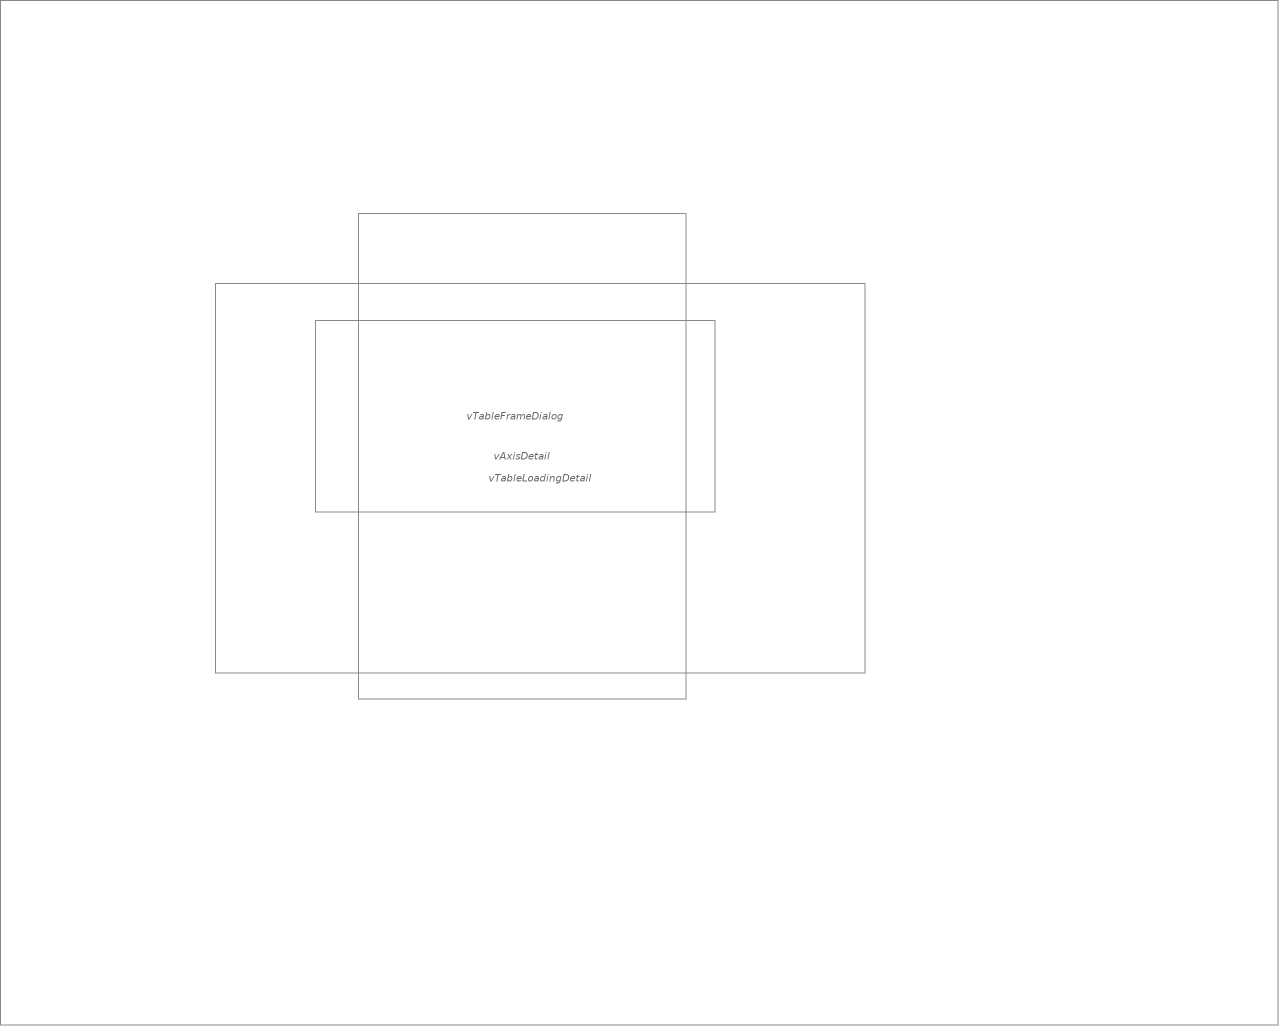
VISUALIZATION vWeighingTunnel  // 1279x1026
VAR_IN_OUT
	fbTableControl: FB_TableControl;
END_VAR
    Rectangle (19,221 146x45), "Drawer Unlock Request", colour toggle: MAIN.fbWeighingStation.bDrawerUnlockRequest, input disabled if: MAIN.fbWeighingStation.stSettings.iMaxNOK_Bottles = MAIN.fbWeighingStation.stSettings.iNOK_BottleCounter
        toggle MAIN.fbWeighingStation.bDrawerUnlockRequest
    Frame (20,4 280x209)
        shows vTableMainControl(fbTableControl := MAIN.fbTableControl)
    Frame (420,796 269x181)
        shows vTableBaseStation(fbStation := MAIN.fbUnloadingStation, fbTableControl := MAIN.fbTableControl)
    Frame (12,370 269x181)
        shows vTableBaseStation(fbStation := MAIN.fbWeighingStation, fbTableControl := MAIN.fbTableControl)
    Frame (489,350 130x210)
        shows vAxisMainParamsDisplay(fbAxis := MAIN.fbTableAxis, fbTableControl := fbTableControl)
    Frame (486,194 137x147)
        shows vTableFrame(fbTablePlace := fbTableControl.arrPlacePositions[1]^, fbTableControl := fbTableControl)
    Frame (341,256 137x147)
        shows vTableFrame(fbTablePlace := fbTableControl.arrPlacePositions[2]^, fbTableControl := fbTableControl)
    Frame (307,411 137x147)
        shows vTableFrame(fbTablePlace := fbTableControl.arrPlacePositions[3]^, fbTableControl := fbTableControl)
    Frame (341,568 137x147)
        shows vTableFrame(fbTablePlace := fbTableControl.arrPlacePositions[4]^, fbTableControl := fbTableControl)
    Frame (486,640 137x147)
        shows vTableFrame(fbTablePlace := fbTableControl.arrPlacePositions[5]^, fbTableControl := fbTableControl)
    Frame (629,568 137x147)
        shows vTableFrame(fbTablePlace := fbTableControl.arrPlacePositions[6]^, fbTableControl := fbTableControl)
    Frame (664,411 137x147)
        shows vTableFrame(fbTablePlace := fbTableControl.arrPlacePositions[7]^, fbTableControl := fbTableControl)
    Frame (629,256 137x147)
        shows vTableFrame(fbTablePlace := fbTableControl.arrPlacePositions[8]^, fbTableControl := fbTableControl)
    Frame (420,4 269x181)
        shows vTableBaseStation(fbStation := MAIN.fbLoadingStation, fbTableControl := MAIN.fbTableControl)
    Rectangle (0,0 1279x1026), invisible if: fbTableControl.stHMI.iDialogNumber=0
    Frame (358,213 328x486), invisible if: fbTableControl.stHMI.iDialogNumber<>100
        shows vAxisDetail(fbAxis := MAIN.fbTableAxis, fbTableControl := MAIN.fbTableControl)
    Frame (215,283 650x390), invisible if: fbTableControl.stHMI.iDialogNumber< 200 OR fbTableControl.stHMI.iDialogNumber >206, frame switch variable: fbTableControl.stHMI.iDialogNumber-200
        shows vTableLoadingDetail(fbStation := MAIN.fbLoadingStation, fbTableControl := fbTableControl)
        shows vTableWeighingDetail(fbStation := MAIN.fbWeighingStation, fbTableControl := fbTableControl)
        shows vTableUnoadingDetail(fbStation := MAIN.fbUnloadingStation, fbTableControl := fbTableControl)
        shows vTableWeighingService(fbStation := MAIN.fbWeighingStation, fbTableControl := fbTableControl)
        shows vTableWeighingWeight(fbStation := MAIN.fbWeighingStation, fbTableControl := fbTableControl)
        shows vTableWeighingVision(fbStation := MAIN.fbWeighingStation, fbTableControl := fbTableControl)
        shows vTableEditTypes(fbTableControl := MAIN.fbTableControl)
    Frame (315,320 400x192), invisible if: fbTableControl.stHMI.iDialogNumber=0 OR fbTableControl.stHMI.iDialogNumber >20
        shows vTableFrameDialog(fbTableControl := fbTableControl)
END_VISUALIZATION

(* stored: Version 1.1.0.1, ProductVersion 3.1.4024.15
   Visu vWeighingTunnel: Id {68710a2b-321f-4eee-82df-79d0b7209949} *)
